// TwinCAT 3 PLC project Untitled1
// ProgramVersion: 3.1.4023.0
// libraries:
//   Tc2_Standard, * (Beckhoff Automation GmbH)
//   Tc2_System, * (Beckhoff Automation GmbH)
//   Tc2_Utilities, * (Beckhoff Automation GmbH)
//   Tc3_Module, * (Beckhoff Automation GmbH)
// project tree:
//   Functions/ Sign.TcPOU (not stored)
//   GVLs/ Param.TcGVL
//   Main Program/ MAIN.TcPOU
//   / PlcTask.TcTTO (not stored)
//   POUs/ DiscreteIntegrator.TcPOU (not stored), ElectricMotor.TcPOU (not stored), HydraulicCylinder.TcPOU, OrificeEquation.TcPOU (not stored), PressureBuildUp.TcPOU, PressureGradient.TcPOU, Pump.TcPOU (not stored)

// ---- GVLs/Param.TcGVL
{attribute 'qualified_only'}
VAR_GLOBAL
	pS : LREAL := 180;
	pT : LREAL := 1;
	BulkModulus : LREAL := 10000;
	Kv : LREAL := 30 / SQRT(7); 
	DBore : LREAL := 60;
	DRod : LREAL := 40;
	xMax : LREAL := 1.5;
	pi : LREAL := 3.14159265359;
    VA0 : LREAL := 0.2;
	VB0 : LREAL := 0.2;

END_VAR

// ---- Main Program/MAIN.TcPOU
PROGRAM MAIN
VAR
	//Integrator
	ssMethodType : SINT := 1; 
	Timer : LREAL;
	
	//Pressure pA
	fbPressureGradient_pA : PressureGradient;
	PressurepA : LREAL;
	
	//Pressure pB
	fbPressureGradient_pB : PressureGradient;
	PressurepB : LREAL;
	
	//Pump
	fbPump : Pump;
	PumpTorque : LREAL;
	PumpFlowRate : LREAL;

	//OrificeEquation QA and QB
	fbOrificeEquationQA : OrificeEquation;
	fbOrificeEquationQB : OrificeEquation;	
	FlowQA : LREAL;
	FlowQB : LREAL;
	
	//HydraulicCylinder
	fbHydraulicCylinder : HydraulicCylinder;
	PressureBoreSide : LREAL;
	PressureRodSide : LREAL;
	AreaBoreSide : LREAL;
	AreaRodSide : LREAL;
	LoadForcePistonFL : LREAL;
	FrictionForce : LREAL;
	PistonMass : LREAL;
	
	pA : LREAL;
	pB : LREAL;
	qA : LREAL;
	qB : LREAL;
	ABore : LREAL;
	ARod : LREAL;
	xPos : LREAL;
	
END_VAR

//Timer
Timer := Timer + 0.01;

//Area Cylinder
ABore := EXPT(Param.DBore,2) * (Param.pi/4.0);
ARod := (EXPT(Param.DBore,2) - EXPT(Param.DRod,2)) * (Param.pi/4.0);

//Pump
fbPump(
	MotorSpeedRPM := 413.2,
	PumpDisplacement := 10.6E-6,
	DeltaMaxPressure := 250.0,
	PumpTorque => PumpTorque,
	PumpFlowRate => PumpFlowRate
	);
	
//Pressure Gradient pA and Pressure pA
fbPressureGradient_pA(
	TotalVolume := 2.9444E-04 + (fbHydraulicCylinder.PistonPosition * fbHydraulicCylinder.AreaBoreSide),
	BulkModulus := 10000.0,
	FlowrateIn := (FlowQA),
	FlowrateOut := (fbHydraulicCylinder.PistonVelocity * fbHydraulicCylinder.AreaBoreSide + 1),
	PressurePascal => PressurepA		//Pressure
	);
	
//Pressure Gradient pB and Pressure pB
fbPressureGradient_pB(
	TotalVolume := 2.9444E-04 + ((1.7 - fbHydraulicCylinder.PistonPosition) * fbHydraulicCylinder.AreaRodSide),
	BulkModulus := 10000.0,
	FlowrateIn := (fbHydraulicCylinder.PistonVelocity * fbHydraulicCylinder.AreaRodSide + 1),
	FlowrateOut := FlowQB,
	PressurePascal => PressurepB		//Pressure
	);


//OrificeEquationA (Q_A)
fbOrificeEquationQA(
	PressureOut := param.pT, 			//Found value from old simulink project, this one goes to the tank i guess
	PressureIn := PressurepA,		
	Kv := 0.5,
	ValveOpening := 1,	
	OrificeFlow => FlowQA
	);
	
//OrificeEquationB (Q_B)
fbOrificeEquationQB(
	PressureOut := param.pT, 			//Found value from old simulink project, this one goes to the tank i guess
	PressureIn := PressurepB,		
	Kv := 0.5,
	ValveOpening := 1,
	OrificeFlow => FlowQB
	);
	
//Hydraulic Cylinder 1
fbHydraulicCylinder(
	PistonMass := 5,
	LoadForcePistonFL := 1,
	FrictionForce := 1,
	AreaBoreSide := ABore,
	AreaRodSide := ARod,
	PressureBoreSide := PressurepA,
	PressureRodSide := PressurepB,
	PistonPosition => xPos
	);

END_PROGRAM

// ---- POUs/PressureGradient.TcPOU
FUNCTION_BLOCK PressureGradient
VAR_INPUT
	TotalVolume: LREAL;
	BulkModulus: LREAL;
	FlowrateIn: LREAL;
	FlowrateOut: LREAL;
END_VAR
VAR_OUTPUT
	PressureGradientBar : LREAL;
	PressureGradientPascal : LREAL;
	PressureBar : LREAL;
	PressurePascal : LREAL;
END_VAR
VAR
	ssMethodType : SINT := 1; 
	fbPressureBar : DiscreteIntegrator;
END_VAR


(* Outputs for Atomic SubSystem: '<Root>/PressureGradient' *)
(* Outport: '<Root>/PressureGradientb' incorporates:
 *  Gain: '<S1>/Conv.2'
 *  Product: '<S1>/Product'
 *  Product: '<S1>/Product1'
 *  Sum: '<S1>/Sum' *)
 
//PressureGradient in [Bar/s]
PressureGradientBar := ((FlowrateIn - FlowrateOut) * 1.6666666666666667E-5) * (Param.BulkModulus / TotalVolume);
(* End of Outputs for SubSystem: '<Root>/PressureGradient' *)

//Multiplies to get [Pascal/s]
PressureGradientPascal := PressureGradientBar*1E5; 

//Pressure in [Pascal]
fbPressureBar(
	ssMethodType := ssMethodType,
	In1 := PressureGradientBar,
	Out1 => PressureBar
	);

//Pressure in [Bar]
PressurePascal := PressureBar*1E5;

END_FUNCTION_BLOCK

// ---- POUs/HydraulicCylinder.TcPOU
FUNCTION_BLOCK HydraulicCylinder
VAR_INPUT
	PressureBoreSide: LREAL;
	PressureRodSide: LREAL;
	AreaBoreSide: LREAL;
	AreaRodSide: LREAL;
	LoadForcePistonFL: LREAL;
	FrictionForce: LREAL;
	PistonMass: LREAL;
END_VAR
VAR_OUTPUT
	PistonAcceleration: LREAL;
	PistonVelocity : LREAL;
	PistonPosition : LREAL;
END_VAR
VAR
	ssMethodType : SINT := 1; 
	fbPistonVelocity : DiscreteIntegrator;
	fbPistonPosition : DiscreteIntegrator;
END_VAR


(* Outputs for Atomic SubSystem: '<Root>/HydraulicCylinder' *)
(* Outport: '<Root>/PistonAcceleration' incorporates:
 *  Gain: '<S1>/Gain1'
 *  Gain: '<S1>/Gain2'
 *  Product: '<S1>/Divide '
 *  Product: '<S1>/Product'
 *  Product: '<S1>/Product1'
 *  Sum: '<S1>/sum' *)
PistonAcceleration := (((((PressureBoreSide * AreaBoreSide) * 100000.0) - ((PressureRodSide * AreaRodSide) * 100000.0)) - FrictionForce) - LoadForcePistonFL) / PistonMass;
(* End of Outputs for SubSystem: '<Root>/HydraulicCylinder' *)

fbPistonVelocity(
	ssMethodType := ssMethodType,
	In1 := PistonAcceleration,
	Out1 => PistonVelocity
	);
	
fbPistonPosition(
	ssMethodType := ssMethodType,
	In1 := PistonVelocity,
	Out1 => PistonPosition
	);

END_FUNCTION_BLOCK

// ---- POUs/PressureBuildUp.TcPOU
FUNCTION_BLOCK PressureBuildUp
VAR
	fbPressureGradient : PressureGradient;
	fbDiscreteIntegrator : DiscreteIntegrator;
	
	IntegratorIn : LREAL;
	IntegratorOut : LREAL;
	ssMethodType : SINT := 1; 
	
//	fbPressure : DiscreteIntegrator;
//	fbPressureGradient : PressureGradient;
END_VAR
VAR_INPUT
	TotalVolume1 : LREAL;
	FlowrateIn1 : LREAL;
	FlowrateOut1 : LREAL;
END_VAR
VAR_OUTPUT
//	PressureBar : LREAL;
//	PressurePascal : LREAL;
END_VAR


fbPressureGradient(
	TotalVolume := TotalVolume1,
	FlowrateIn := FlowrateIn1,
	FlowrateOut := FlowrateOut1
	);

//pA
(* fbPressure(
	ssMethodType := ssMethodType,
	In1 := fbPressureGradient.PressureGradientPascal,
	Out1 => PressurePascal
	);
	
PressureGradientPascal := PressureGradientBar*1E5;      //Multiplies to get Pascal *)

END_FUNCTION_BLOCK
